screen "02_Parametros_Ecu" 800x447, template "Template_1"
   IOField "I/O field_1" at 46,125 size 154x33; FormatPattern 99999999999999999999
      ProcessValue <- "DB303_ScadaToCentral_Data_Turnos_Inicio{0}"
   TextField "Text field_1" at 63,98 size 115x20; Text 'Inicio de Turno'
   TextField "Text field_2" at 68,162 size 98x20; Text 'Fim de Turno'
   IOField "I/O field_3" at 46,244 size 150x33; FormatPattern 999999
      ProcessValue <- "DB303_ScadaToCentral_Data_ParametrosTakt{0}_Tempo_Takt"
   TextField "Text field_3" at 63,222 size 112x20; Text 'Tempo de Takt'
   IOField "I/O field_4" at 46,297 size 149x33; FormatPattern 999999
      ProcessValue <- "DB303_ScadaToCentral_Data_ParametrosTakt{0}_ObjetivoTurno"
   TextField "Text field_4" at 52,277 size 136x20; Text 'Objetivo do turno'
   Button "Button_1" at 61,334 size 116x32; TextOff 'PARADAS PROGRAMADAS'
      on Release: ActivateScreen("03_Paradas_1Turno", 0)
   Button "Button_4" at 7,19 size 88x30; TextOff 'HOME'
      on Release: ActivateScreen("01_Home", 0)
   TextField "Text field_13" at 216,18 size 352x25; Text 'Parametros do TAKT Powertrain-ECU'
   IOField "I/O field_5" at 45,188 size 154x33; FormatPattern 99999999999999999999
      ProcessValue <- "DB303_ScadaToCentral_Data_Turnos_Fim{0}"
   TextField "Text field_5" at 56,70 size 131x22; Text 'Primeiro Turno'
   IOField "I/O field_2" at 312,125 size 154x33; FormatPattern 99999999999999999999
      ProcessValue <- "DB303_ScadaToCentral_Data_Turnos_Inicio{1}"
   TextField "Text field_6" at 329,98 size 115x20; Text 'Inicio de Turno'
   TextField "Text field_7" at 334,162 size 98x20; Text 'Fim de Turno'
   IOField "I/O field_6" at 312,243 size 150x33; FormatPattern 999999
      ProcessValue <- "DB303_ScadaToCentral_Data_ParametrosTakt{1}_Tempo_Takt"
   TextField "Text field_8" at 329,224 size 112x20; Text 'Tempo de Takt'
   IOField "I/O field_7" at 312,298 size 149x33; FormatPattern 999999
      ProcessValue <- "DB303_ScadaToCentral_Data_ParametrosTakt{1}_ObjetivoTurno"
   TextField "Text field_9" at 318,277 size 136x20; Text 'Objetivo do turno'
   Button "Button_2" at 327,336 size 116x32; TextOff 'PARADAS PROGRAMADAS'
      on Release: ActivateScreen("03_Paradas_1Turno", 0)
   IOField "I/O field_8" at 311,188 size 154x33; FormatPattern 99999999999999999999
      ProcessValue <- "DB303_ScadaToCentral_Data_Turnos_Fim{1}"
   TextField "Text field_10" at 322,70 size 129x22; Text 'Segunda Turno'
   IOField "I/O field_9" at 578,125 size 154x33; FormatPattern 99999999999999999999
      ProcessValue <- "DB303_ScadaToCentral_Data_Turnos_Inicio{2}"
   TextField "Text field_11" at 595,98 size 115x20; Text 'Inicio de Turno'
   TextField "Text field_12" at 600,162 size 98x20; Text 'Fim de Turno'
   IOField "I/O field_10" at 578,243 size 150x33; FormatPattern 999999
      ProcessValue <- "DB303_ScadaToCentral_Data_ParametrosTakt{2}_Tempo_Takt"
   TextField "Text field_14" at 595,225 size 112x20; Text 'Tempo de Takt'
   IOField "I/O field_11" at 578,294 size 149x33; FormatPattern 999999
      ProcessValue <- "DB303_ScadaToCentral_Data_ParametrosTakt{2}_ObjetivoTurno"
   TextField "Text field_15" at 584,276 size 136x20; Text 'Objetivo do turno'
   Button "Button_3" at 593,331 size 116x32; TextOff 'PARADAS PROGRAMADAS'
      on Release: ActivateScreen("03_Paradas_1Turno", 0)
   IOField "I/O field_12" at 577,188 size 154x33; FormatPattern 99999999999999999999
      ProcessValue <- "DB303_ScadaToCentral_Data_Turnos_Fim{2}"
   TextField "Text field_16" at 588,70 size 129x22; Text 'Terceiro Turno'
   Switch "Switch_1" at 659,7 size 136x52; CaptionText 'Input Takt'; TextOff 'IHM'; TextOn 'SISTEMA'
      on SwitchOn: SetBit("DB302_InputDados_Ecu_SistemaOn")
      on SwitchOff: ResetBit("DB302_InputDados_Ecu_SistemaOn")
      ProcessValue <- "DB302_InputDados_Ecu_SistemaOn"
   Switch "Switch_2" at 15,394 size 104x46; CaptionText 'Segunda-feira'; TextOff 'OFF'; TextOn 'ON'
      on SwitchOn: SetBit("DB303_ScadaToCentral_Data_Dias_Da_Semana{0}")
      on SwitchOff: ResetBit("DB303_ScadaToCentral_Data_Dias_Da_Semana{0}")
      ProcessValue <- "DB303_ScadaToCentral_Data_Dias_Da_Semana{0}"
   Switch "Switch_3" at 123,394 size 104x46; TextOn 'ON'; CaptionText 'Terça-feira'; TextOff 'OFF'
      on SwitchOff: ResetBit("DB303_ScadaToCentral_Data_Dias_Da_Semana{1}")
      on SwitchOn: SetBit("DB303_ScadaToCentral_Data_Dias_Da_Semana{1}")
      ProcessValue <- "DB303_ScadaToCentral_Data_Dias_Da_Semana{1}"
   Switch "Switch_4" at 232,394 size 104x46; TextOn 'ON'; CaptionText 'Quarta-feira'; TextOff 'OFF'
      on SwitchOff: ResetBit("DB303_ScadaToCentral_Data_Dias_Da_Semana{2}")
      on SwitchOn: SetBit("DB303_ScadaToCentral_Data_Dias_Da_Semana{2}")
      ProcessValue <- "DB303_ScadaToCentral_Data_Dias_Da_Semana{2}"
   Switch "Switch_5" at 341,394 size 104x46; TextOn 'ON'; CaptionText 'Quinta-feira'; TextOff 'OFF'
      on SwitchOff: ResetBit("DB303_ScadaToCentral_Data_Dias_Da_Semana{3}")
      on SwitchOn: SetBit("DB303_ScadaToCentral_Data_Dias_Da_Semana{3}")
      ProcessValue <- "DB303_ScadaToCentral_Data_Dias_Da_Semana{3}"
   Switch "Switch_6" at 449,394 size 104x46; TextOn 'ON'; CaptionText 'Sexta-feira'; TextOff 'OFF'
      on SwitchOff: ResetBit("DB303_ScadaToCentral_Data_Dias_Da_Semana{4}")
      on SwitchOn: SetBit("DB303_ScadaToCentral_Data_Dias_Da_Semana{4}")
      ProcessValue <- "DB303_ScadaToCentral_Data_Dias_Da_Semana{4}"
   Switch "Switch_7" at 558,394 size 104x46; TextOn 'ON'; CaptionText 'Sabado'; TextOff 'OFF'
      on SwitchOff: ResetBit("DB303_ScadaToCentral_Data_Dias_Da_Semana{5}")
      on SwitchOn: SetBit("DB303_ScadaToCentral_Data_Dias_Da_Semana{5}")
      ProcessValue <- "DB303_ScadaToCentral_Data_Dias_Da_Semana{5}"
   Switch "Switch_8" at 669,394 size 104x46; TextOn 'ON'; CaptionText 'Domingo'; TextOff 'OFF'
      on SwitchOff: ResetBit("DB303_ScadaToCentral_Data_Dias_Da_Semana{6}")
      on SwitchOn: SetBit("DB303_ScadaToCentral_Data_Dias_Da_Semana{6}")
      ProcessValue <- "DB303_ScadaToCentral_Data_Dias_Da_Semana{6}"

screen "02_Parametros_Cab" 800x447, template "Template_1"
   IOField "I/O field_1" at 46,125 size 154x33; FormatPattern 9999999999999999999999999999999999999999
      ProcessValue <- "DB302_InputDados_Cabinas_Turnos_1_Turno_Inicio"
   TextField "Text field_1" at 63,98 size 115x20; Text 'Inicio de Turno'
   TextField "Text field_2" at 68,162 size 98x20; Text 'Fim de Turno'
   IOField "I/O field_3" at 46,260 size 150x33; FormatPattern 999999
      ProcessValue <- "DB302_InputDados_Cabinas_Turnos_1_Turno_TempoTakt"
   TextField "Text field_3" at 63,230 size 112x20; Text 'Tempo de Takt'
   IOField "I/O field_4" at 46,334 size 149x33; FormatPattern 999999
      ProcessValue <- "DB302_InputDados_Cabinas_Turnos_1_Turno_Rodadas"
   TextField "Text field_4" at 52,304 size 136x20; Text 'Objetivo do turno'
   Button "Button_1" at 61,382 size 116x32; TextOff 'PARADAS PROGRAMADAS'
   Button "Button_4" at 7,19 size 88x30; TextOff 'HOME'
      on Release: ActivateScreen("01_Home", 0)
   TextField "Text field_13" at 244,16 size 322x25; Text 'Parametros do TAKT Cabinas-ECU'
   IOField "I/O field_5" at 45,188 size 154x33; FormatPattern 9999999999999999999999999999999999999999
      ProcessValue <- "DB302_InputDados_Cabinas_Turnos_1_Turno_Fim"
   TextField "Text field_5" at 56,70 size 131x22; Text 'Primeiro Turno'
   IOField "I/O field_2" at 312,125 size 154x33; FormatPattern 9999999999999999999999999999999999999999
      ProcessValue <- "DB302_InputDados_Cabinas_Turnos_2_Turno_Inicio"
   TextField "Text field_6" at 329,98 size 115x20; Text 'Inicio de Turno'
   TextField "Text field_7" at 334,162 size 98x20; Text 'Fim de Turno'
   IOField "I/O field_6" at 312,260 size 150x33; FormatPattern 999999
      ProcessValue <- "DB302_InputDados_Cabinas_Turnos_2_Turno_TempoTakt"
   TextField "Text field_8" at 329,230 size 112x20; Text 'Tempo de Takt'
   IOField "I/O field_7" at 312,334 size 149x33; FormatPattern 999999
      ProcessValue <- "DB302_InputDados_Cabinas_Turnos_2_Turno_Rodadas"
   TextField "Text field_9" at 318,304 size 136x20; Text 'Objetivo do turno'
   Button "Button_2" at 327,382 size 116x32; TextOff 'PARADAS PROGRAMADAS'
   IOField "I/O field_8" at 311,188 size 154x33; FormatPattern 9999999999999999999999999999999999999999
      ProcessValue <- "DB302_InputDados_Cabinas_Turnos_2_Turno_Fim"
   TextField "Text field_10" at 322,70 size 129x22; Text 'Segunda Turno'
   IOField "I/O field_9" at 578,125 size 154x33; FormatPattern 9999999999999999999999999999999999999999
      ProcessValue <- "DB302_InputDados_Cabinas_Turnos_3_Turno_Inicio"
   TextField "Text field_11" at 595,98 size 115x20; Text 'Inicio de Turno'
   TextField "Text field_12" at 600,162 size 98x20; Text 'Fim de Turno'
   IOField "I/O field_10" at 578,260 size 150x33; FormatPattern 999999
      ProcessValue <- "DB302_InputDados_Cabinas_Turnos_3_Turno_TempoTakt"
   TextField "Text field_14" at 595,230 size 112x20; Text 'Tempo de Takt'
   IOField "I/O field_11" at 578,334 size 149x33; FormatPattern 999999
      ProcessValue <- "DB302_InputDados_Cabinas_Turnos_3_Turno_Rodadas"
   TextField "Text field_15" at 584,304 size 136x20; Text 'Objetivo do turno'
   Button "Button_3" at 593,382 size 116x32; TextOff 'PARADAS PROGRAMADAS'
   IOField "I/O field_12" at 577,188 size 154x33; FormatPattern 9999999999999999999999999999999999999999
      ProcessValue <- "DB302_InputDados_Cabinas_Turnos_3_Turno_Fim"
   TextField "Text field_16" at 588,70 size 129x22; Text 'Terceiro Turno'
   Switch "Switch_1" at 659,7 size 136x52; TextOn 'SISTEMA'; CaptionText 'Input Takt'; TextOff 'IHM'
      on SwitchOn: SetBit("DB302_InputDados_Cabinas_SistemaOn")
      on SwitchOff: ResetBit("DB302_InputDados_Cabinas_SistemaOn")
      ProcessValue <- "DB302_InputDados_Cabinas_SistemaOn"

screen "02_Parametros_Skd" 800x447, template "Template_1"
   IOField "I/O field_1" at 50,122 size 154x33; FormatPattern 9999999999999999999999999999999999999999
      ProcessValue <- "DB302_InputDados_SKD_Turnos_1_Turno_Inicio"
   TextField "Text field_1" at 67,95 size 115x20; Text 'Inicio de Turno'
   TextField "Text field_2" at 72,159 size 98x20; Text 'Fim de Turno'
   IOField "I/O field_3" at 50,257 size 150x33; FormatPattern 999999
      ProcessValue <- "DB302_InputDados_SKD_Turnos_1_Turno_TempoTakt"
   TextField "Text field_3" at 67,227 size 112x20; Text 'Tempo de Takt'
   IOField "I/O field_4" at 50,331 size 149x33; FormatPattern 999999
      ProcessValue <- "DB302_InputDados_SKD_Turnos_1_Turno_Rodadas"
   TextField "Text field_4" at 56,301 size 136x20; Text 'Objetivo do turno'
   Button "Button_1" at 65,379 size 116x32; TextOff 'PARADAS PROGRAMADAS'
   Button "Button_4" at 11,16 size 88x30; TextOff 'HOME'
      on Release: ActivateScreen("01_Home", 0)
   TextField "Text field_13" at 272,16 size 242x25; Text 'Parametros do TAKT SKD'
   IOField "I/O field_5" at 49,185 size 154x33; FormatPattern 9999999999999999999999999999999999999999
      ProcessValue <- "DB302_InputDados_SKD_Turnos_1_Turno_Fim"
   TextField "Text field_5" at 60,67 size 131x22; Text 'Primeiro Turno'
   IOField "I/O field_2" at 316,122 size 154x33; FormatPattern 9999999999999999999999999999999999999999
      ProcessValue <- "DB302_InputDados_SKD_Turnos_2_Turno_Inicio"
   TextField "Text field_6" at 333,95 size 115x20; Text 'Inicio de Turno'
   TextField "Text field_7" at 338,159 size 98x20; Text 'Fim de Turno'
   IOField "I/O field_6" at 316,257 size 150x33; FormatPattern 999999
      ProcessValue <- "DB302_InputDados_SKD_Turnos_2_Turno_TempoTakt"
   TextField "Text field_8" at 333,227 size 112x20; Text 'Tempo de Takt'
   IOField "I/O field_7" at 316,331 size 149x33; FormatPattern 999999
      ProcessValue <- "DB302_InputDados_SKD_Turnos_2_Turno_Rodadas"
   TextField "Text field_9" at 322,301 size 136x20; Text 'Objetivo do turno'
   Button "Button_2" at 331,379 size 116x32; TextOff 'PARADAS PROGRAMADAS'
   IOField "I/O field_8" at 315,185 size 154x33; FormatPattern 9999999999999999999999999999999999999999
      ProcessValue <- "DB302_InputDados_SKD_Turnos_2_Turno_Fim"
   TextField "Text field_10" at 326,67 size 129x22; Text 'Segunda Turno'
   IOField "I/O field_9" at 582,122 size 154x33; FormatPattern 9999999999999999999999999999999999999999
      ProcessValue <- "DB302_InputDados_SKD_Turnos_3_Turno_Inicio"
   TextField "Text field_11" at 599,95 size 115x20; Text 'Inicio de Turno'
   TextField "Text field_12" at 604,159 size 98x20; Text 'Fim de Turno'
   IOField "I/O field_10" at 582,257 size 150x33; FormatPattern 999999
      ProcessValue <- "DB302_InputDados_SKD_Turnos_3_Turno_TempoTakt"
   TextField "Text field_14" at 599,227 size 112x20; Text 'Tempo de Takt'
   IOField "I/O field_11" at 582,331 size 149x33; FormatPattern 999999
      ProcessValue <- "DB302_InputDados_SKD_Turnos_3_Turno_Rodadas"
   TextField "Text field_15" at 588,301 size 136x20; Text 'Objetivo do turno'
   Button "Button_3" at 597,379 size 116x32; TextOff 'PARADAS PROGRAMADAS'
   IOField "I/O field_12" at 581,185 size 154x33; FormatPattern 9999999999999999999999999999999999999999
      ProcessValue <- "DB302_InputDados_SKD_Turnos_3_Turno_Fim"
   TextField "Text field_16" at 592,67 size 129x22; Text 'Terceiro Turno'
   Switch "Switch_1" at 659,7 size 136x52; TextOn 'SISTEMA'; CaptionText 'Input Takt'; TextOff 'IHM'
      on SwitchOn: SetBit("DB302_InputDados_SKD_SistemaOn")
      on SwitchOff: ResetBit("DB302_InputDados_SKD_SistemaOn")
      ProcessValue <- "DB302_InputDados_SKD_SistemaOn"

screen "02_Parametros_Comp" 800x447, template "Template_1"
   IOField "I/O field_1" at 55,127 size 154x33; FormatPattern 9999999999999999999999999999999999999999
      ProcessValue <- "DB302_InputDados_Componentes_Turnos_1_Turno_Inicio"
   TextField "Text field_1" at 72,100 size 115x20; Text 'Inicio de Turno'
   TextField "Text field_2" at 77,164 size 98x20; Text 'Fim de Turno'
   IOField "I/O field_3" at 55,262 size 150x33; FormatPattern 999999
      ProcessValue <- "DB302_InputDados_Componentes_Turnos_1_Turno_TempoTakt"
   TextField "Text field_3" at 72,232 size 112x20; Text 'Tempo de Takt'
   IOField "I/O field_4" at 55,336 size 149x33; FormatPattern 999999
      ProcessValue <- "DB302_InputDados_Componentes_Turnos_1_Turno_Rodadas"
   TextField "Text field_4" at 61,306 size 136x20; Text 'Objetivo do turno'
   Button "Button_1" at 70,384 size 116x32; TextOff 'PARADAS PROGRAMADAS'
   Button "Button_4" at 16,14 size 88x30; TextOff 'HOME'
      on Release: ActivateScreen("01_Home", 0)
   TextField "Text field_13" at 211,13 size 444x25; Text 'Parametros do TAKT Powertrain-Componentes'
   IOField "I/O field_5" at 54,190 size 154x33; FormatPattern 9999999999999999999999999999999999999999
      ProcessValue <- "DB302_InputDados_Componentes_Turnos_1_Turno_Fim"
   TextField "Text field_5" at 65,72 size 131x22; Text 'Primeiro Turno'
   IOField "I/O field_2" at 321,127 size 154x33; FormatPattern 9999999999999999999999999999999999999999
      ProcessValue <- "DB302_InputDados_Componentes_Turnos_2_Turno_Inicio"
   TextField "Text field_6" at 338,100 size 115x20; Text 'Inicio de Turno'
   TextField "Text field_7" at 343,164 size 98x20; Text 'Fim de Turno'
   IOField "I/O field_6" at 321,262 size 150x33; FormatPattern 999999
      ProcessValue <- "DB302_InputDados_Componentes_Turnos_2_Turno_TempoTakt"
   TextField "Text field_8" at 338,232 size 112x20; Text 'Tempo de Takt'
   IOField "I/O field_7" at 321,336 size 149x33; FormatPattern 999999
      ProcessValue <- "DB302_InputDados_Componentes_Turnos_2_Turno_Rodadas"
   TextField "Text field_9" at 327,306 size 136x20; Text 'Objetivo do turno'
   Button "Button_2" at 336,384 size 116x32; TextOff 'PARADAS PROGRAMADAS'
   IOField "I/O field_8" at 320,190 size 154x33; FormatPattern 9999999999999999999999999999999999999999
      ProcessValue <- "DB302_InputDados_Componentes_Turnos_2_Turno_Fim"
   TextField "Text field_10" at 331,72 size 129x22; Text 'Segunda Turno'
   IOField "I/O field_9" at 587,127 size 154x33; FormatPattern 9999999999999999999999999999999999999999
      ProcessValue <- "DB302_InputDados_Componentes_Turnos_3_Turno_Inicio"
   TextField "Text field_11" at 604,100 size 115x20; Text 'Inicio de Turno'
   TextField "Text field_12" at 609,164 size 98x20; Text 'Fim de Turno'
   IOField "I/O field_10" at 587,262 size 150x33; FormatPattern 999999
      ProcessValue <- "DB302_InputDados_Componentes_Turnos_3_Turno_TempoTakt"
   TextField "Text field_14" at 604,232 size 112x20; Text 'Tempo de Takt'
   IOField "I/O field_11" at 587,336 size 149x33; FormatPattern 999999
      ProcessValue <- "DB302_InputDados_Componentes_Turnos_3_Turno_Rodadas"
   TextField "Text field_15" at 593,306 size 136x20; Text 'Objetivo do turno'
   Button "Button_3" at 602,384 size 116x32; TextOff 'PARADAS PROGRAMADAS'
   IOField "I/O field_12" at 586,190 size 154x33; FormatPattern 9999999999999999999999999999999999999999
      ProcessValue <- "DB302_InputDados_Componentes_Turnos_3_Turno_Fim"
   TextField "Text field_16" at 597,72 size 129x22; Text 'Terceiro Turno'
   Switch "Switch_1" at 659,7 size 136x52; TextOn 'SISTEMA'; CaptionText 'Input Takt'; TextOff 'IHM'
      ProcessValue <- "DB302_InputDados_Componentes_SistemaOn"

screen "03_Paradas_1Turno" 800x447, template "Template_1"
   IOField "I/O field_1" at 52,111 size 109x34; FormatPattern 9999999999999999999999999999999999999999
      ProcessValue <- "DB303_ScadaToCentral_Data_Paradas_Programadas_Inicio{0}"
   TextField "Text field_1" at 45,88 size 125x20; Text 'Inicio da Parada'
   IOField "I/O field_2" at 52,172 size 109x34; FormatPattern 9999999999999999999999999999999999999999
      ProcessValue <- "DB303_ScadaToCentral_Data_Paradas_Programadas_Fim{0}"
   TextField "Text field_2" at 52,149 size 108x20; Text 'Fim da Parada'
   IOField "I/O field_3" at 336,111 size 109x34; FormatPattern 9999999999999999999999999999999999999999
      ProcessValue <- "DB303_ScadaToCentral_Data_Paradas_Programadas_Inicio{1}"
   TextField "Text field_3" at 329,88 size 125x20; Text 'Inicio da Parada'
   IOField "I/O field_4" at 336,172 size 109x34; FormatPattern 9999999999999999999999999999999999999999
      ProcessValue <- "DB303_ScadaToCentral_Data_Paradas_Programadas_Fim{1}"
   TextField "Text field_4" at 336,149 size 108x20; Text 'Fim da Parada'
   IOField "I/O field_5" at 620,111 size 109x34; FormatPattern 9999999999999999999999999999999999999999
      ProcessValue <- "DB303_ScadaToCentral_Data_Paradas_Programadas_Inicio{2}"
   TextField "Text field_5" at 613,88 size 125x20; Text 'Inicio da Parada'
   IOField "I/O field_6" at 620,172 size 109x34; FormatPattern 9999999999999999999999999999999999999999
      ProcessValue <- "DB303_ScadaToCentral_Data_Paradas_Programadas_Fim{2}"
   TextField "Text field_6" at 620,149 size 108x20; Text 'Fim da Parada'
   IOField "I/O field_7" at 191,303 size 109x34; FormatPattern 99999999999999999999
      ProcessValue <- "DB303_ScadaToCentral_Data_Paradas_Programadas_Inicio{4}"
   TextField "Text field_7" at 184,280 size 125x20; Text 'Inicio da Parada'
   IOField "I/O field_8" at 191,364 size 109x34; FormatPattern 99999999999999999999
      ProcessValue <- "DB303_ScadaToCentral_Data_Paradas_Programadas_Fim{4}"
   TextField "Text field_8" at 191,341 size 108x20; Text 'Fim da Parada'
   IOField "I/O field_9" at 479,303 size 109x34; FormatPattern 99999999999999999999
      ProcessValue <- "DB303_ScadaToCentral_Data_Paradas_Programadas_Inicio{5}"
   TextField "Text field_9" at 472,280 size 125x20; Text 'Inicio da Parada'
   IOField "I/O field_10" at 479,364 size 109x34; FormatPattern 99999999999999999999
      ProcessValue <- "DB303_ScadaToCentral_Data_Paradas_Programadas_Fim{5}"
   TextField "Text field_10" at 479,341 size 108x20; Text 'Fim da Parada'
   TextField "Text field_11" at 52,57 size 115x20; Text 'Parada Almoço'
   TextField "Text field_12" at 323,57 size 165x20; Text 'Parada Programada 1'
   TextField "Text field_13" at 607,57 size 165x20; Text 'Parada Programada 2'
   TextField "Text field_14" at 178,252 size 165x20; Text 'Parada Programada 3'
   TextField "Text field_15" at 466,252 size 165x20; Text 'Parada Programada 4'
   Button "Button_4" at 7,19 size 88x30; TextOff 'VOLTAR'
      on Release: ActivateScreen("02_Parametros_Ecu", 0)
   TextField "Text field_16" at 178,19 size 510x25; Text 'Paradas programadas para o Powertrain-ECU 1 Turno'

screen "04_Paradas_2Turno" 800x447, template "Template_1"
   IOField "I/O field_1" at 52,111 size 109x34; FormatPattern 99999999999999999999
      ProcessValue <- "DB302_InputDados_Ecu_Paradas_Programadas_2Turno_Parada_1_Inicio"
   TextField "Text field_1" at 45,88 size 125x20; Text 'Inicio da Parada'
   IOField "I/O field_2" at 52,172 size 109x34; FormatPattern 99999999999999999999
      ProcessValue <- "DB302_InputDados_Ecu_Paradas_Programadas_2Turno_Parada_1_Fim"
   TextField "Text field_2" at 52,149 size 108x20; Text 'Fim da Parada'
   IOField "I/O field_3" at 336,111 size 109x34; FormatPattern 99999999999999999999
      ProcessValue <- "DB302_InputDados_Ecu_Paradas_Programadas_2Turno_Parada_2_Inicio"
   TextField "Text field_3" at 329,88 size 125x20; Text 'Inicio da Parada'
   IOField "I/O field_4" at 336,172 size 109x34; FormatPattern 99999999999999999999
      ProcessValue <- "DB302_InputDados_Ecu_Paradas_Programadas_2Turno_Parada_2_Fim"
   TextField "Text field_4" at 336,149 size 108x20; Text 'Fim da Parada'
   IOField "I/O field_5" at 620,111 size 109x34; FormatPattern 99999999999999999999
      ProcessValue <- "DB302_InputDados_Ecu_Paradas_Programadas_2Turno_Parada_3_Inicio"
   TextField "Text field_5" at 613,88 size 125x20; Text 'Inicio da Parada'
   IOField "I/O field_6" at 620,172 size 109x34; FormatPattern 99999999999999999999
      ProcessValue <- "DB302_InputDados_Ecu_Paradas_Programadas_2Turno_Parada_3_Fim"
   TextField "Text field_6" at 620,149 size 108x20; Text 'Fim da Parada'
   IOField "I/O field_7" at 191,303 size 109x34; FormatPattern 99999999999999999999
      ProcessValue <- "DB302_InputDados_Ecu_Paradas_Programadas_2Turno_Parada_4_Inicio"
   TextField "Text field_7" at 184,280 size 125x20; Text 'Inicio da Parada'
   IOField "I/O field_8" at 191,364 size 109x34; FormatPattern 99999999999999999999
      ProcessValue <- "DB302_InputDados_Ecu_Paradas_Programadas_2Turno_Parada_4_Fim"
   TextField "Text field_8" at 191,341 size 108x20; Text 'Fim da Parada'
   IOField "I/O field_9" at 479,303 size 109x34; FormatPattern 99999999999999999999
      ProcessValue <- "DB302_InputDados_Ecu_Paradas_Programadas_2Turno_Parada_5_Inicio"
   TextField "Text field_9" at 472,280 size 125x20; Text 'Inicio da Parada'
   IOField "I/O field_10" at 479,364 size 109x34; FormatPattern 99999999999999999999
      ProcessValue <- "DB302_InputDados_Ecu_Paradas_Programadas_2Turno_Parada_5_Fim"
   TextField "Text field_10" at 479,341 size 108x20; Text 'Fim da Parada'
   TextField "Text field_11" at 52,57 size 103x20; Text 'Parada Janta'
   TextField "Text field_12" at 323,57 size 165x20; Text 'Parada Programada 1'
   TextField "Text field_13" at 607,57 size 165x20; Text 'Parada Programada 2'
   TextField "Text field_14" at 178,252 size 165x20; Text 'Parada Programada 3'
   TextField "Text field_15" at 466,252 size 165x20; Text 'Parada Programada 4'
   Button "Button_4" at 7,19 size 88x30; TextOff 'VOLTAR'
      on Release: ActivateScreen("02_Parametros_Ecu", 0)
   TextField "Text field_16" at 182,17 size 510x25; Text 'Paradas programadas para o Powertrain-ECU 2 Turno'

screen "05_Paradas_3Turno" 800x447, template "Template_1"
   IOField "I/O field_1" at 52,111 size 109x34; FormatPattern 99999999999999999999
      ProcessValue <- "DB302_InputDados_Ecu_Paradas_Programadas_3Turno_Parada_1_Inicio"
   TextField "Text field_1" at 45,88 size 125x20; Text 'Inicio da Parada'
   IOField "I/O field_2" at 52,172 size 109x34; FormatPattern 99999999999999999999
      ProcessValue <- "DB302_InputDados_Ecu_Paradas_Programadas_3Turno_Parada_1_Fim"
   TextField "Text field_2" at 52,149 size 108x20; Text 'Fim da Parada'
   IOField "I/O field_3" at 336,111 size 109x34; FormatPattern 99999999999999999999
      ProcessValue <- "DB302_InputDados_Ecu_Paradas_Programadas_3Turno_Parada_2_Inicio"
   TextField "Text field_3" at 329,88 size 125x20; Text 'Inicio da Parada'
   IOField "I/O field_4" at 336,172 size 109x34; FormatPattern 99999999999999999999
      ProcessValue <- "DB302_InputDados_Ecu_Paradas_Programadas_3Turno_Parada_2_Fim"
   TextField "Text field_4" at 336,149 size 108x20; Text 'Fim da Parada'
   IOField "I/O field_5" at 620,111 size 109x34; FormatPattern 99999999999999999999
      ProcessValue <- "DB302_InputDados_Ecu_Paradas_Programadas_3Turno_Parada_3_Inicio"
   TextField "Text field_5" at 613,88 size 125x20; Text 'Inicio da Parada'
   IOField "I/O field_6" at 620,172 size 109x34; FormatPattern 99999999999999999999
      ProcessValue <- "DB302_InputDados_Ecu_Paradas_Programadas_3Turno_Parada_3_Fim"
   TextField "Text field_6" at 620,149 size 108x20; Text 'Fim da Parada'
   IOField "I/O field_7" at 191,303 size 109x34; FormatPattern 99999999999999999999
      ProcessValue <- "DB302_InputDados_Ecu_Paradas_Programadas_3Turno_Parada_4_Inicio"
   TextField "Text field_7" at 184,280 size 125x20; Text 'Inicio da Parada'
   IOField "I/O field_8" at 191,364 size 109x34; FormatPattern 99999999999999999999
      ProcessValue <- "DB302_InputDados_Ecu_Paradas_Programadas_3Turno_Parada_4_Fim"
   TextField "Text field_8" at 191,341 size 108x20; Text 'Fim da Parada'
   IOField "I/O field_9" at 479,303 size 109x34; FormatPattern 99999999999999999999
      ProcessValue <- "DB302_InputDados_Ecu_Paradas_Programadas_3Turno_Parada_5_Inicio"
   TextField "Text field_9" at 472,280 size 125x20; Text 'Inicio da Parada'
   IOField "I/O field_10" at 479,364 size 109x34; FormatPattern 99999999999999999999
      ProcessValue <- "DB302_InputDados_Ecu_Paradas_Programadas_3Turno_Parada_5_Fim"
   TextField "Text field_10" at 479,341 size 108x20; Text 'Fim da Parada'
   TextField "Text field_11" at 52,57 size 95x20; Text 'Parada Café'
   TextField "Text field_12" at 323,57 size 165x20; Text 'Parada Programada 1'
   TextField "Text field_13" at 607,57 size 165x20; Text 'Parada Programada 2'
   TextField "Text field_14" at 178,252 size 165x20; Text 'Parada Programada 3'
   TextField "Text field_15" at 466,252 size 165x20; Text 'Parada Programada 4'
   Button "Button_4" at 7,19 size 88x30; TextOff 'VOLTAR'
      on Release: ActivateScreen("02_Parametros_Ecu", 0)
   TextField "Text field_16" at 173,18 size 510x25; Text 'Paradas programadas para o Powertrain-ECU 3 Turno'

screen "06_StatusDeAndon" 800x447, template "Template_1"
   Button "Button_4" at 7,19 size 88x30; TextOff 'VOLTAR'
      on Release: ActivateScreen("01_Home", 0)
   TextField "Text field_16" at 216,19 size 447x25; Text 'Status dos andons da linha de Powertrain-ECU'

screen "07_UltimasParadas" 800x447, template "Template_1"
   Button "Button_4" at 7,19 size 88x30; TextOff 'VOLTAR'
      on Release: ActivateScreen("01_Home", 0)
   TextField "Text field_16" at 216,19 size 424x25; Text 'Ultimas paradas na linha de Powertrain-ECU'

VB script "TitleUpdater"
   Dim title
   Set title = HmiRuntime.Screens(0).ScreenItems("Screen title")
   title.Text = HmiRuntime.BaseScreenName

VB script "VBFunction_1"
   'Tip:
   ' 1. Use the <CTRL+SPACE> or <CTRL+I> shortcut to open a list of all objects and functions
   ' 2. Write the code using the HMI Runtime object.
   '  Example: HmiRuntime.Screens("Screen_1").
   ' 3. Use the <CTRL+J> shortcut to create an object reference.
   'Write the code as of this position:
*)